FUNCTION_BLOCK TestFB EXTENDS SignalHandling
VAR_INPUT
	rTemperature : REAL;
END_VAR
VAR_OUTPUT
END_VAR
VAR
	bLowPressure : BOOL;
	bWaitForRelease : BOOL;
END_VAR

SUPER^();

IF rTemperature = 0 
THEN
	Throw(BuildException(eWRONG_VALUE_EXCEPTION));	
END_IF

IF bLowPressure
THEN
	Throw(BuildException(eLOW_PRESSURE_EXCEPTION));
END_IF

IF bWaitForRelease
THEN
	bWaitForRelease := FALSE;
	Signal(BuildSignal(eWAIT_FOR_RELEASE_SIGNAL));
END_IF

END_FUNCTION_BLOCK

(* stored: Version 1.1.0.1, ProductVersion 3.1.4024.0
   POU TestFB: Id {e7ed8dd4-ef00-486c-9202-c82c305437bc}, SpecialFunc None *)
